PROGRAM P_BACnet_Error
VAR
	i					: INT := 0;		//for loop counter
	arrLampFailure		: ARRAY [1..10] OF BOOL;
	dwLampFailure		: DWORD;
	rLampFailure		: REAL;
	
	fbDALIV2QueryLampFailure_1		: FB_DALIV2QueryLampFailure;
	fbDALIV2QueryLampFailure_2		: FB_DALIV2QueryLampFailure;
END_VAR

//iterate through DALI ballasts reading lamp failure information
FOR i := 1 TO byStreetLampsCount BY 1 DO
	//query first half of the lamp
	fbDALIV2QueryLampFailure_1(
			bStart:= TRUE, 
			nAddr:= GVL_IO.arrStreetLamps[i].nAddrShort1, 
			eAddrType:= eDALIV2AddrTypeShort, 
			eCommandPriority:= eDALIV2CommandPriorityLow,  
			stCommandBuffer:= GVL_IO.arrStreetLamps[i].ref_stCommandBuffer);
	//reset the block
	fbDALIV2QueryLampFailure_1(bStart := FALSE, stCommandBuffer := GVL_IO.arrStreetLamps[i].ref_stCommandBuffer);

	//query second half of the lamp
	fbDALIV2QueryLampFailure_2(
			bStart:= TRUE, 
			nAddr:= GVL_IO.arrStreetLamps[i].nAddrShort2, 
			eAddrType:= eDALIV2AddrTypeShort, 
			eCommandPriority:= eDALIV2CommandPriorityLow,  
			stCommandBuffer:= GVL_IO.arrStreetLamps[i].ref_stCommandBuffer);
	//reset the block
	fbDALIV2QueryLampFailure_2(bStart := FALSE, stCommandBuffer := GVL_IO.arrStreetLamps[i].ref_stCommandBuffer);
	
	
	//if at least one of ballasts indicates failure, set flag (LampFailure) to TRUE
	arrLampFailure[i] := fbDALIV2QueryLampFailure_1.bLampFailure OR fbDALIV2QueryLampFailure_2.bLampFailure;	
END_FOR
		
//convert arrLampFailure into pseudo-array in the form of a DWORD variable
dwLampFailure.0 := arrLampFailure[1];
dwLampFailure.1 := arrLampFailure[2];
dwLampFailure.2 := arrLampFailure[3];
dwLampFailure.3 := arrLampFailure[4];
dwLampFailure.4 := arrLampFailure[5];
dwLampFailure.5 := arrLampFailure[6];
dwLampFailure.6 := arrLampFailure[7];
dwLampFailure.7 := arrLampFailure[8];
dwLampFailure.8 := arrLampFailure[9];
dwLampFailure.9 := arrLampFailure[10];

//type conversion from REAL to DWORD
rLampFailure := DWORD_TO_REAL(dwLampFailure);

//write rLampFailure to BACnet obcject present value
//thereby keep BACnet object instance alive
fbBACnet_AV_SL_Error(Device := Device, bEnablePV := TRUE, bNullPV := FALSE, fPV := rLampFailure);

END_PROGRAM

(* stored: Version 1.1.0.1, ProductVersion 3.1.4024.5
   POU P_BACnet_Error: Id {cbcb446d-2870-4188-9eca-74baf4a350e8}, SpecialFunc None *)
